// TIA Portal V21 export
TYPE "UDT_ Caja"
   STRUCT
      Alta : Bool;
      Baja : Bool;
   END_STRUCT;
END_TYPE
